FUNCTION_BLOCK FB_CycleAuto
(**)
VAR_INPUT
	xStart			:BOOL; (*start input command*)
	//xStopCmdPin			:BOOL; (*stop input command*)
	xReset			:BOOL; (*Reset input command*)
		(*Station index*)
	
END_VAR
VAR_OUTPUT
	xDone			:BOOL;(*Done output*)
	xBusy				:BOOL;(*Busy output*)
END_VAR
VAR_IN_OUT
	//fbErrorAdmin:FB_ErrorAdmin;
END_VAR
VAR
	

	iStep			: INT;		(* cycle step *)
	iNextStep			: INT;		(* cycle step *)
	fbTrigStart			: R_Trig;	(*Trigger for start*)
	fbTimerTON			:TON;
	
END_VAR

(*Reset  if xReset is set to true*)
IF xReset
	THEN
		xReset:=FALSE;
		iStep:=0;
		xDone:=FALSE;
END_IF

fbTrigStart(CLK:=xStart);


CASE  iStep OF
	0:	IF fbTrigStart.Q
		THEN
		xDone:=FALSE;
		iStep:=100;
		END_IF
	
	100: fbStation.fbAxeX.fbMoveAbsolute.Position:=GVL.stParam.stRecipe.lrPositionBasse;
			fbStation.fbAxeX.fbMoveAbsolute.Velocity:=GVL.stParam.stRecipe.lrVitesse;
			iStep:=200;
			
	200: IF  fbStation.fbAxeX.fbMoveAbsolute.Done
		THEN
			iStep:=250;
	END_IF
	
	250:  fbStation.fbAxeX.fbMoveAbsolute.Position:=0;
			fbStation.fbAxeX.fbMoveAbsolute.Velocity:=GVL.stParam.stRecipe.lrVitesse;
			iStep:=300;
			
	300: IF  fbStation.fbAxeX.fbMoveAbsolute.Done
		THEN
			iStep:=900;
	END_IF

	900: xDone:=TRUE;
		iStep:=0;

END_CASE

fbTimerTON(IN:=iStep=210);
xBusy:=iStep<>0;

END_FUNCTION_BLOCK

(* stored: Version 1.1.0.1, ProductVersion 3.1.4020.12
   POU FB_CycleAuto: Id {276925a8-9c19-4dad-9bb7-674fd1b013cf}, SpecialFunc None *)
